FUNCTION_BLOCK FB_Main
VAR_INPUT
END_VAR
VAR_OUTPUT
END_VAR
VAR
// Areas
	s_unMachine	: FB_Area100;
END_VAR

// Areas
s_unMachine();

END_FUNCTION_BLOCK

(* stored: Version 1.1.0.1, ProductVersion 3.1.4026.13
   POU FB_Main: Id {ce4e8b74-9023-48c1-875b-79162c03d5fc}, SpecialFunc None *)
